DATA_BLOCK "Valves"
{ S7_Optimized_Access := 'FALSE' }
VERSION : 0.1
   STRUCT
      V001 : "VState";
      V002 : "VState";
      V003 : "VState";
      V008 : "VState";
      V009 : "VState";
      V012 : "VState";
      V057 : "VState";
      V058 : "VState";
      V059 : "VState";
      V060 : "VState";
      V061 : "VState";
      V063 : "VState";
      V064 : "VState";
      V070 : "VState";
      V071 : "VState";
      V072 : "VState";
      V073 : "VState";
      V074 : "VState";
      V075 : "VState";
      V076 : "VState";
      V077 : "VState";
      V078 : "VState";
      V079 : "VState";
      V080 : "VState";
   END_STRUCT;


BEGIN
   V001.IsAuto := TRUE;
   V001.Close := TRUE;
   V001.countOpening := BYTE#16#05;
   V001.countClosing := BYTE#16#05;
   V002.IsAuto := TRUE;
   V002.Close := TRUE;
   V002.countOpening := BYTE#16#05;
   V002.countClosing := BYTE#16#05;
   V003.IsAuto := TRUE;
   V003.Close := TRUE;
   V003.countOpening := BYTE#16#05;
   V003.countClosing := BYTE#16#05;
   V008.IsAuto := TRUE;
   V008.Close := TRUE;
   V008.countOpening := BYTE#16#05;
   V008.countClosing := BYTE#16#05;
   V009.IsAuto := TRUE;
   V009.Close := TRUE;
   V009.countOpening := BYTE#16#05;
   V009.countClosing := BYTE#16#05;
   V012.IsAuto := TRUE;
   V012.Close := TRUE;
   V012.countOpening := BYTE#16#05;
   V012.countClosing := BYTE#16#05;
   V057.IsAuto := TRUE;
   V057.Close := TRUE;
   V057.countOpening := BYTE#16#05;
   V057.countClosing := BYTE#16#05;
   V058.IsAuto := TRUE;
   V058.Close := TRUE;
   V058.countOpening := BYTE#16#05;
   V058.countClosing := BYTE#16#05;
   V059.IsAuto := TRUE;
   V059.Close := TRUE;
   V059.countOpening := BYTE#16#05;
   V059.countClosing := BYTE#16#05;
   V060.IsAuto := TRUE;
   V060.Close := TRUE;
   V060.countOpening := BYTE#16#05;
   V060.countClosing := BYTE#16#05;
   V061.IsAuto := TRUE;
   V061.Close := TRUE;
   V061.countOpening := BYTE#16#05;
   V061.countClosing := BYTE#16#05;
   V063.IsAuto := TRUE;
   V063.Close := TRUE;
   V063.countOpening := BYTE#16#05;
   V063.countClosing := BYTE#16#05;
   V064.IsAuto := TRUE;
   V064.Close := TRUE;
   V064.countOpening := BYTE#16#05;
   V064.countClosing := BYTE#16#05;
   V070.IsAuto := TRUE;
   V070.Close := TRUE;
   V070.countOpening := BYTE#16#05;
   V070.countClosing := BYTE#16#05;
   V071.IsAuto := TRUE;
   V071.Close := TRUE;
   V071.countOpening := BYTE#16#05;
   V071.countClosing := BYTE#16#05;
   V072.IsAuto := TRUE;
   V072.Close := TRUE;
   V072.countOpening := BYTE#16#05;
   V072.countClosing := BYTE#16#05;
   V073.IsAuto := TRUE;
   V073.Close := TRUE;
   V073.countOpening := BYTE#16#05;
   V073.countClosing := BYTE#16#05;
   V074.IsAuto := TRUE;
   V074.Close := TRUE;
   V074.countOpening := BYTE#16#05;
   V074.countClosing := BYTE#16#05;
   V075.IsAuto := TRUE;
   V075.Close := TRUE;
   V075.countOpening := BYTE#16#05;
   V075.countClosing := BYTE#16#05;
   V076.IsAuto := TRUE;
   V076.Close := TRUE;
   V076.countOpening := BYTE#16#05;
   V076.countClosing := BYTE#16#05;
   V077.IsAuto := TRUE;
   V077.Close := TRUE;
   V077.countOpening := BYTE#16#05;
   V077.countClosing := BYTE#16#05;
   V078.IsAuto := TRUE;
   V078.Close := TRUE;
   V078.countOpening := BYTE#16#05;
   V078.countClosing := BYTE#16#05;
   V079.IsAuto := TRUE;
   V079.Close := TRUE;
   V079.countOpening := BYTE#16#05;
   V079.countClosing := BYTE#16#05;
   V080.IsAuto := TRUE;
   V080.Close := TRUE;
   V080.countOpening := BYTE#16#05;
   V080.countClosing := BYTE#16#05;

END_DATA_BLOCK

